SYSTEM VAV_VIEWL (* Variable Air Valve System View+HMI *)
  (* Standard: 61499-1; Classification: Simulation; ApplicationDomain: HVAC *)
  (* Version 0.1, 2007-03-29, JHC, Holobloc Inc, Made ROOM_REND tag usage consistent. *)
  (* Version 0.0, 2006-04-06, JHC, Holobloc Inc *)
  DEVICE RECORDER : FRAME_DEVICE(BOUNDS := [240,100,210,250])
    RESOURCE RECORDER : PANEL_RESOURCE
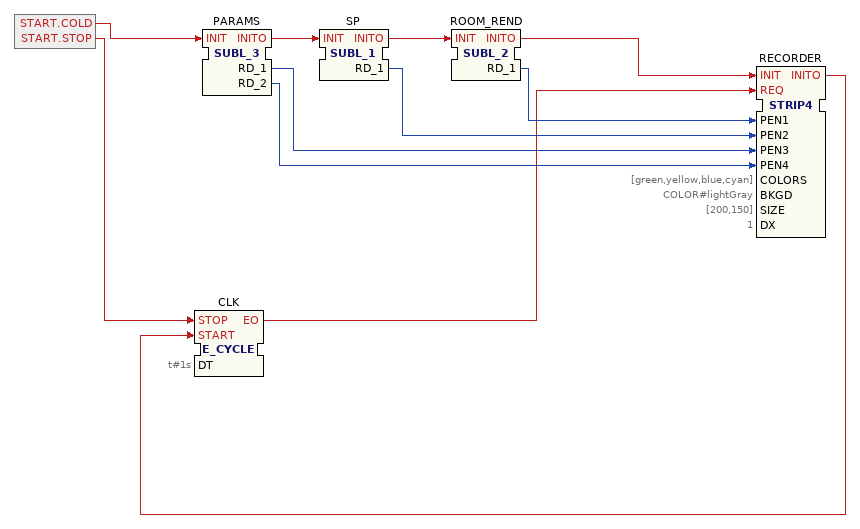
      FBS
        RECORDER : STRIP4(COLORS := [green,yellow,blue,cyan], BKGD := COLOR#lightGray, SIZE := [200,150], DX := 1);
        SP : SUBL_1;
        PARAMS : SUBL_3;
        ROOM_REND : SUBL_2;
        CLK : E_CYCLE(DT := t#1s);
      END_FBS
      EVENT_CONNECTIONS
        START.COLD TO PARAMS.INIT;
        PARAMS.INITO TO SP.INIT;
        SP.INITO TO ROOM_REND.INIT;
        ROOM_REND.INITO TO RECORDER.INIT;
        START.STOP TO CLK.STOP;
        RECORDER.INITO TO CLK.START;
        CLK.EO TO RECORDER.REQ;
      END_CONNECTIONS
      DATA_CONNECTIONS
        ROOM_REND.RD_1 TO RECORDER.PEN1;
        SP.RD_1 TO RECORDER.PEN2;
        PARAMS.RD_1 TO RECORDER.PEN3;
        PARAMS.RD_2 TO RECORDER.PEN4;
      END_CONNECTIONS
    END_RESOURCE
    RESOURCE PARAMS : PANEL_RESOURCE(ROWS := 2, COLS := 2)
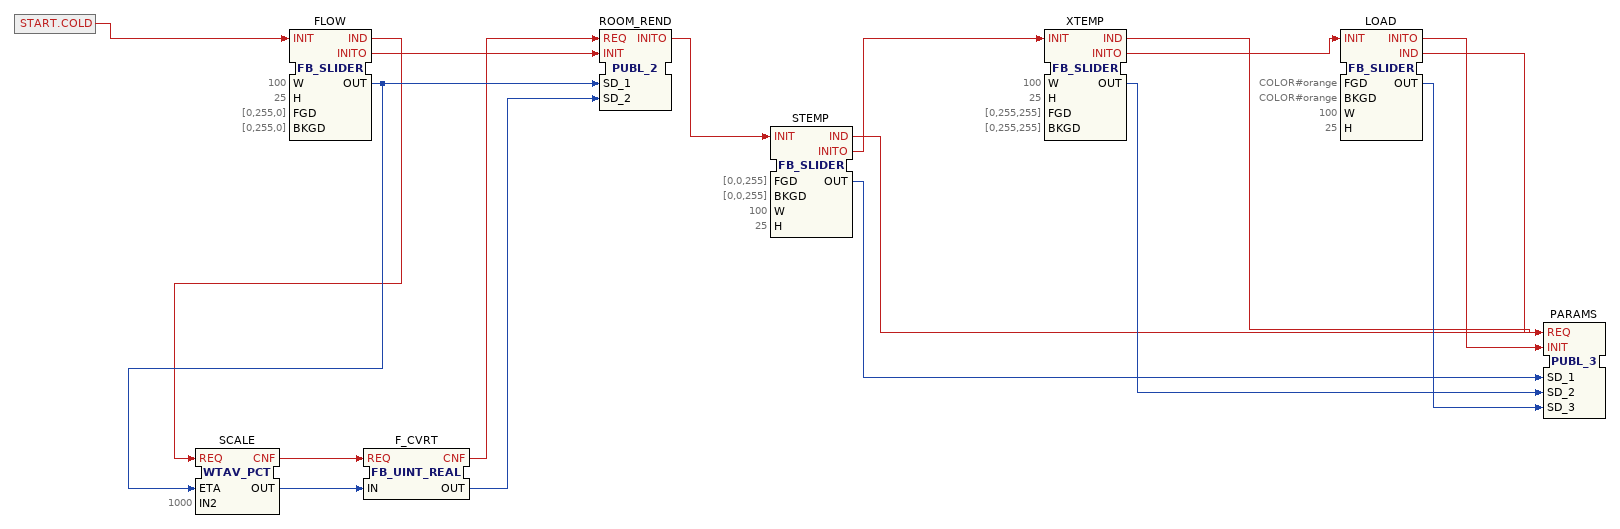
      FBS
        PARAMS : PUBL_3;
        FLOW : FB_SLIDER(W := 100, H := 25, FGD := [0,255,0], BKGD := [0,255,0]);
        STEMP : FB_SLIDER(FGD := [0,0,255], BKGD := [0,0,255], W := 100, H := 25);
        XTEMP : FB_SLIDER(W := 100, H := 25, FGD := [0,255,255], BKGD := [0,255,255]);
        LOAD : FB_SLIDER(FGD := COLOR#orange, BKGD := COLOR#orange, W := 100, H := 25);
        SCALE : WTAV_PCT(IN2 := 1000);
        F_CVRT : FB_UINT_REAL;
        ROOM_REND : PUBL_2;
      END_FBS
      EVENT_CONNECTIONS
        START.COLD TO FLOW.INIT;
        STEMP.IND TO PARAMS.REQ;
        STEMP.INITO TO XTEMP.INIT;
        XTEMP.IND TO PARAMS.REQ;
        XTEMP.INITO TO LOAD.INIT;
        LOAD.INITO TO PARAMS.INIT;
        LOAD.IND TO PARAMS.REQ;
        F_CVRT.CNF TO ROOM_REND.REQ;
        FLOW.IND TO SCALE.REQ;
        SCALE.CNF TO F_CVRT.REQ;
        FLOW.INITO TO ROOM_REND.INIT;
        ROOM_REND.INITO TO STEMP.INIT;
      END_CONNECTIONS
      DATA_CONNECTIONS
        FLOW.OUT TO ROOM_REND.SD_1;
        STEMP.OUT TO PARAMS.SD_1;
        XTEMP.OUT TO PARAMS.SD_2;
        LOAD.OUT TO PARAMS.SD_3;
        F_CVRT.OUT TO ROOM_REND.SD_2;
        FLOW.OUT TO SCALE.ETA;
        SCALE.OUT TO F_CVRT.IN;
      END_CONNECTIONS
    END_RESOURCE
  END_DEVICE
  DEVICE CTRL : FRAME_DEVICE(BOUNDS := [100,100,140,270])
    RESOURCE FACE : PANEL_RESOURCE
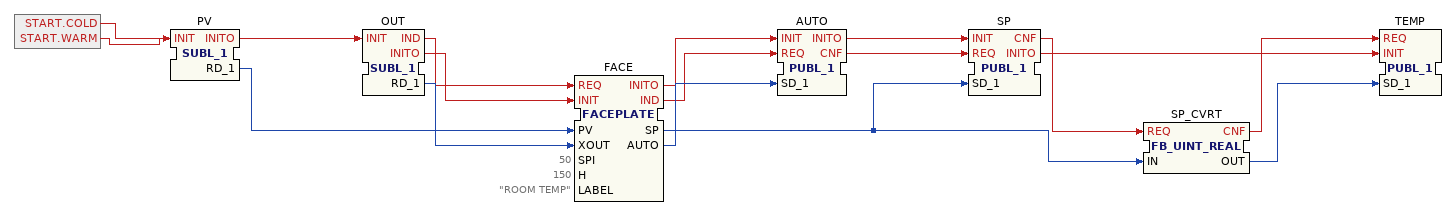
      FBS
        PV : SUBL_1;
        FACE : FACEPLATE(SPI := 50, H := 150, LABEL := "ROOM TEMP");
        SP : PUBL_1;
        OUT : SUBL_1;
        AUTO : PUBL_1;
        TEMP : PUBL_1;
        SP_CVRT : FB_UINT_REAL;
      END_FBS
      EVENT_CONNECTIONS
        START.COLD TO PV.INIT;
        START.WARM TO PV.INIT;
        OUT.IND TO FACE.REQ;
        FACE.INITO TO AUTO.INIT;
        FACE.IND TO AUTO.REQ;
        AUTO.INITO TO SP.INIT;
        AUTO.CNF TO SP.REQ;
        PV.INITO TO OUT.INIT;
        OUT.INITO TO FACE.INIT;
        SP.CNF TO SP_CVRT.REQ;
        SP_CVRT.CNF TO TEMP.REQ;
        SP.INITO TO TEMP.INIT;
      END_CONNECTIONS
      DATA_CONNECTIONS
        PV.RD_1 TO FACE.PV;
        FACE.SP TO SP.SD_1;
        OUT.RD_1 TO FACE.XOUT;
        FACE.AUTO TO AUTO.SD_1;
        SP_CVRT.OUT TO TEMP.SD_1;
        FACE.SP TO SP_CVRT.IN;
      END_CONNECTIONS
    END_RESOURCE
  END_DEVICE
  DEVICE VIEW : FRAME_DEVICE(BOUNDS := [450,100,290,250])
    RESOURCE DUCTS : VIEW_PANEL(DIA := 25, SIZE := [3,8], VERTICAL := 1)
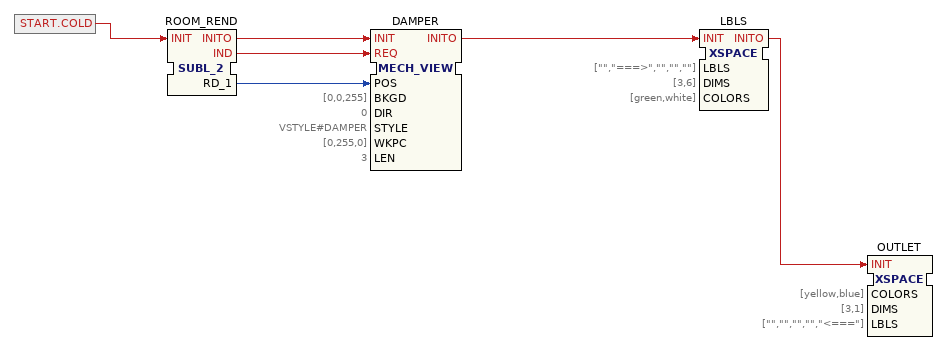
      FBS
        ROOM_REND : SUBL_2;
        DAMPER : MECH_VIEW(BKGD := [0,0,255], DIR := 0, STYLE := VSTYLE#DAMPER, WKPC := [0,255,0], LEN := 3);
        LBLS : XSPACE(LBLS := ["","===>","","",""], DIMS := [3,6], COLORS := [green,white]);
        OUTLET : XSPACE(COLORS := [yellow,blue], DIMS := [3,1], LBLS := ["","","","","<==="]);
      END_FBS
      EVENT_CONNECTIONS
        START.COLD TO ROOM_REND.INIT;
        ROOM_REND.INITO TO DAMPER.INIT;
        ROOM_REND.IND TO DAMPER.REQ;
        LBLS.INITO TO OUTLET.INIT;
        DAMPER.INITO TO LBLS.INIT;
      END_CONNECTIONS
      DATA_CONNECTIONS
        ROOM_REND.RD_1 TO DAMPER.POS;
      END_CONNECTIONS
    END_RESOURCE
    RESOURCE ROOM : VIEW_PANEL(SIZE := [8,8], DIA := 25)
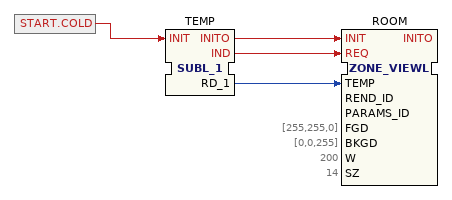
      FBS
        ROOM : ZONE_VIEWL(FGD := [255,255,0], BKGD := [0,0,255], W := 200, SZ := 14);
        TEMP : SUBL_1;
      END_FBS
      EVENT_CONNECTIONS
        START.COLD TO TEMP.INIT;
        TEMP.INITO TO ROOM.INIT;
        TEMP.IND TO ROOM.REQ;
      END_CONNECTIONS
      DATA_CONNECTIONS
        TEMP.RD_1 TO ROOM.TEMP;
      END_CONNECTIONS
    END_RESOURCE
  END_DEVICE
END_SYSTEM
